3:
	(* 	Clamp State Machine 														*)
	(*		Init: TS back, collets unclamped, ejectors Retracted, Unclamped				*)
	(*		T0: Clamp Requested													*)
	(*		S1: a) Advance Tailstock to Forward Position 				 				*)
	(*			b) When collett significantly swallows part Advance Ejectors. Start Timer	*)
	(*		T1: Tailstock @ Forward Position										*)
	(*		S2: Verify  Ejectors Status of Advanced Proxes and Time Delay completed		*)
	(*		T2: Ejectors Advanced Confirmation 										*)
	(*		S3: Clamp Collet 														*)
	(*		T3: All Report Clamped PS 												*)
	(*		S4: Turn Off Postion Lag Monitoring and Set Torque Limit Value				*)
	(*		T4: Confirm Donef														*)
	(*		S5: Issue Move Velocity (in proper direction)								*)
	(*		T5: Verify Torque Value												*)
	(*		S6: REPORT CLAMPED 												*)
	IF NOT(bEnable) THEN
		bColletClamp:=FALSE;
		bColletUnclamp:=FALSE;
		bEjectorAdvance:=FALSE;
		bEjectorRetract:=FALSE;
		bTailstockAxisMove:=FALSE;
		bTailstockAxisMoveVelo:=FALSE;
		bEjectorAdvanceTON:=FALSE;
		bColletClampTON:= FALSE;
		bEjectorRetractTON:= FALSE;
		bColletUnclampTON:= FALSE;
		bTailstockAxisStop:=TRUE;
		nCurrentAction:=0;
		nClampingState:=0;
	END_IF
	IF NOT(bClampParts) THEN
		(* WE ONLY GET HERE IF THERE IS AN EXTERNAL FAULT *)
		(* Stop ALL Possible Movement *)
		bEjectorAdvance:=FALSE;
		bEjectorRetract:=FALSE;
		bColletClamp:=FALSE;
		bColletUnclamp:=FALSE;
		bEjectorAdvanceTON:=FALSE;
		bColletClampTON:= FALSE;
		bEjectorRetractTON:= FALSE;
		bColletUnclampTON:= FALSE;
		(* Stop Axis *)
		IF NOT(bTailstockAxisStop) THEN
			bTailstockAxisMove:=FALSE;
			bTailstockAxisMoveVelo:=FALSE;
			bTailstockAxisSetZero:=FALSE;
			bTailstockAxisStop:=TRUE;
		ELSIF bTailstockAxisStop AND fbTailstockAxisStop.Error THEN
			bTailstockAxisStop:=FALSE;
			(* EXIT *)
			nCurrentAction:=2;
			nClampingState:=0;
		ELSIF bTailstockAxisStop AND fbTailstockAxisStop.Done THEN
			bTailstockAxisStop:=FALSE;
			(* EXIT *)
			nCurrentAction:=2;
			nClampingState:=0;
		END_IF
	ELSE
		CASE nClampingState OF
		0:	(* Init: TS back, Parts Ready to Clamp, collets unclamped, Ejectors Retracted, Unclamped *)
			IF bClamped THEN
				nCurrentAction:=2;
			ELSIF stTailstockAxis.NcToPlc.ActPos < fTailstockBackPosition - 0.1 THEN
				nErrorID:=12;
				bError:=TRUE;
				nClampingState:=0;
				nCurrentAction:=255;
			ELSIF NOT(bColletUnclamped) THEN
				nErrorID:=13;
				bError:=TRUE;
				nClampingState:=0;
				nCurrentAction:=255;
			ELSIF NOT(stTailstockAxis.Status.Homed) THEN
				nErrorID:=1;
				bError:=TRUE;
				nClampingState:=0;
				nCurrentAction:=255;
			ELSIF NOT bTransferAtClampPosition THEN
				nErrorID:=14;
				bError:=TRUE;
				nClampingState:=0;
				nCurrentAction:=255;
			ELSIF NOT(nEjectorRetracted=7) THEN
				nErrorID:=15;
				bError:=TRUE;
				nClampingState:=0;
				nCurrentAction:=255;
			(* Begin Clamping *)
			ELSE
			(* T0: Clamp Requested *)
				(* When we are behind the transfer position we move fast to the transfer position *)
				IF (stTailstockAxis.NcToPlc.ActPos > fTailstockFrontPosition + 0.5) THEN
					nClampingState:=7;
				(* When we are at the transfer position we move at the slow speed to swallow the parts *)
				ELSE
					nClampingState:=nClampingState+1;
				END_IF
			END_IF

		1:	(* S1: a) Advance Tailstock to Forward Position
				b) When collett significantly swallows part Advance Ejectors. Start Timer *)
			IF bTailstockAxisMove AND fbTailstockAxisMoveTo.Error THEN
				bTailstockAxisMove:=FALSE;
				bTailstockAxisStop:=TRUE;
				(* Error *)
				nErrorID:=3;
				bError:=TRUE;
				nClampingState:=0;
				nCurrentAction:=255;
			(* When the Torque exceeds Max set value exit and fault *)
			ELSIF nTorqueFeedback>nClampingMaxTorqueLimit*10 THEN
				bTailstockAxisMove:=FALSE;
				bTailstockAxisStop:=TRUE;
				bError:=TRUE;
				nErrorID:=2;
				nClampingState:=0;
				nCurrentAction:=255;
			ELSIF bTailstockAxisMove AND fbTailstockAxisMoveTo.Done AND fbEjectorAdvanceTon.Q THEN
			(* T1: Tailstock @ Position *)
				bTailstockAxisMove:=FALSE;
				nClampingState:=nClampingState+1;
			ELSIF (stTailstockAxis.NcToPlc.ActPos < fTailstockFrontPosition + 8.0) THEN
			 (* S1:b) Advanced Ejectors when significantly swallowed part *)
				bEjectorAdvance:=TRUE;
			ELSE
				fTailstockAxisPosition:=fTailstockFrontPosition;
				fTailstockAxisVelocityLocal:=fTailstockAxisVelocityClamp;
				bTailstockAxisMove:=TRUE;
				(* Turn off the Retract output so the coil field can collapse before we fire other solenoid valve *)
				bEjectorRetract := FALSE;
			END_IF

		2:	(* S2: Verify  Ejectors Status of Advanced Proxes *)
			(* Fault if one of the ejectors overtraveled *)
			IF nEjectorAdvanced<7 AND nEjectorRetracted=0 AND bEjectorAdvance THEN
				(* Error *)
				nErrorID:=5;
				bError:=TRUE;
				nCurrentAction:=255;
				nClampingState:=0;
				bEjectorAdvance:=FALSE;
				bEjectorAdvanceTON:=FALSE;
			(* Basically this step gives the Ejectors a 1/2 second time delay to operate *)
			ELSIF nEjectorAdvanced=7 AND nEjectorRetracted=0 AND bEjectorAdvance  THEN
			(* T2: Ejectors Advanced *)
				nClampingState:=nClampingState+1;
			END_IF

		3:	(* S3: Clamp Collet *)
			IF bColletClamp AND fbColletClampTON.Q THEN
				(* Error *)
				nErrorID:=6;
				bError:=TRUE;
				nCurrentAction:=255;
				nClampingState:=0;
				bColletClamp:=FALSE;
				bColletClampTON:=FALSE;
			(* We look for Ejector Advanced Error in this step in case one of the Ejectors was slow *)
			ELSIF nEjectorAdvanced<7 AND nEjectorRetracted=0 AND bEjectorAdvance THEN
				(* Error *)
				nErrorID:=5;
				bError:=TRUE;
				nCurrentAction:=255;
				nClampingState:=0;
				bEjectorAdvance:=FALSE;
			ELSIF bColletClamped AND bColletClamp THEN
			(* T3: All Report Clamped *)
				bColletClampTON:=FALSE;
				nClampingState:=6;
			ELSE
				bColletUnclamp:=FALSE;
				bColletClampTON:=TRUE;
				(* Allow Solenoid to De-energize before firing Oposing Solenoid *)
				IF fbUnclampOffTON.Q THEN
					bColletClamp:=TRUE;
				END_IF
			END_IF

		(* We were unable to accomplish Torque limited move because the Ejectors overcame the Collet clamping force *)
		4:	(*S4: Turn Off Postion Lag Monitoring AND Set Torque LIMIT Value *)
			nTorqueLimit := nTorqueLimitRequest;
			IF bTogglePositionLagMonitoring AND fbTogglePositionLagMonitoring.Error THEN
				(* Error *)
				nErrorID:=20;
				bError:=TRUE;
				nCurrentAction:=255;
				nClampingState:=0;
				bTogglePositionLagMonitoring:=FALSE;
			ELSIF bTogglePositionLagMonitoring AND fbTogglePositionLagMonitoring.Done  THEN
			(* T4: Done *)
				bTogglePositionLagMonitoring:=FALSE;
				nClampingState:=nClampingState+1;
			ELSE
				bTogglePositionLagMonitoring := TRUE;
				bPositionLagMonitoiring := FALSE;
			END_IF

		5:	(* S5: Issue Move Velocity (in proper direction) *)
			IF bTailstockAxisMoveVelo AND fbTailstockAxisMoveVelo.Error
			THEN
				nVeloMoveErrorID:=fbTailstockAxisMoveVelo.ErrorID;
				bTailstockAxisMoveVelo :=FALSE;
				bTorqueLimitTimeout:=FALSE;
				bTailstockAxisStop := TRUE;
				(* Error *)
				nErrorID:=19;
				bError:=TRUE;
				nClampingState:=0;
				nCurrentAction:=255;
			ELSIF bTailstockAxisMoveVelo AND fbTorqueLimitTON.Q
			THEN
				bTailstockAxisMoveVelo :=FALSE;
				bTorqueLimitTimeout:=FALSE;
				bTailstockAxisStop := TRUE;
				(* Error *)
				nErrorID:=18;
				bError:=TRUE;
				nClampingState:=0;
				nCurrentAction:=255;
			ELSIF bTailstockAxisMoveVelo AND
				(stTailstockAxis.NcToPlc.ActPos < (fTailstockFrontPosition -0.10))
			THEN
				bTailstockAxisMoveVelo :=FALSE;
				bTorqueLimitTimeout:=FALSE;
				bTailstockAxisStop := TRUE;
				(* Error *)
				nErrorID:=17;
				bError:=TRUE;
				nClampingState:=0;
				nCurrentAction:=255;
			ELSIF bTailstockAxisMoveVelo AND (nTorqueFeedback > ( nTorqueLimitRequest - 2 )) THEN
			(* T7: In Velocity Command *)
				bTorqueLimitTimeout:=FALSE;
				bTailstockAxisMoveVelo := FALSE;
				nClampingState:=nClampingState+1;
			ELSE
				fTailstockAxisPosition:=fTailstockFrontPosition+fTailstockAxisBackOffAmount;
				fTailstockMoveVelo:=fTailstockAxisVelocity;
				bTailstockAxisMoveVelo:=TRUE;
				bTorqueLimitTimeout := TRUE;
			END_IF

		6:	(* S6: REPORT CLAMPED *)
			nClampingState:=0;
			nCurrentAction:=2;

		7:	(* Advance to Transfer position *)
			IF bTailstockAxisMove AND fbTailstockAxisMoveTo.Error THEN
				bTailstockAxisMove:=FALSE;
				bTailstockAxisStop:=TRUE;
				(* Error *)
				nErrorID:=3;
				bError:=TRUE;
				nClampingState:=0;
				nCurrentAction:=255;
			(* When the Torque exceeds Max set value exit and fault *)
			ELSIF nTorqueFeedback>nMaxFastTorqueLimit*10 THEN
				bTailstockAxisMove:=FALSE;
				bTailstockAxisStop:=TRUE;
				bError:=TRUE;
				nErrorID:=2;
				nClampingState:=0;
				nCurrentAction:=255;
			ELSIF bTailstockAxisMove AND fbTailstockAxisMoveTo.Done THEN
			(* T1: Tailstock @ Transfer Position *)
				bTailstockAxisMove:=FALSE;
				nClampingState:=1;
			ELSE
				fTailstockAxisPosition:=fTailstockBackPosition;
				fTailstockAxisVelocityLocal:=fTailstockAxisVelocity;
				bTailstockAxisMove:=TRUE;
			END_IF

		END_CASE
	END_IF

4:
	(*	Unclamp State Machine													*)
	(*		Init: All report clamped and reporting clamped								*)
	(*		T0: Unclamp Requested												*)
	(*		S1: Stop Axis															*)
	(*		T1: Done bit															*)
	(*		S2: Set Torque Back to 100%											*)
	(*		S3: Retract Tailstock Offset Amount and Retract Ejectors 						*)
	(*		T3: Tailstock @ Offset 													*)
	(*		S4: Unclamp Collets													*)
	(*		T4: Collets Unclamp PS												*)
	(*		S5: Move Tailstock to back position										*)
	(*		T5: Tailstock @ back 													*)
	(*		S6: REPORT UNCLAMPED												*)

	IF NOT(bEnable) THEN
		bColletClamp:=FALSE;
		bColletUnclamp:=FALSE;
		bEjectorAdvance:=FALSE;
		bEjectorRetract:=FALSE;
		bTailstockAxisMove:=FALSE;
		bEjectorAdvanceTON:=FALSE;
		bColletClampTON:= FALSE;
		bEjectorRetractTON:= FALSE;
		bColletUnclampTON:= FALSE;
		bTailstockAxisStop:=TRUE;
		nCurrentAction:=0;
		nUnclampingState:=0;
	END_IF
	IF NOT(bUnclampParts) THEN
		(* WE ONLY GET HERE IF THERE IS AN EXTERNAL FAULT *)
		(* Stop ALL Possible Movement *)
		bEjectorAdvance:=FALSE;
		bEjectorRetract:=FALSE;
		bColletClamp:=FALSE;
		bColletUnclamp:=FALSE;
		bEjectorAdvanceTON:=FALSE;
		bColletClampTON:= FALSE;
		bEjectorRetractTON:= FALSE;
		bColletUnclampTON:= FALSE;
		(* Stop Axis *)
		IF NOT(bTailstockAxisStop) THEN
			bTailstockAxisHome:=FALSE;
			bTailstockAxisMove:=FALSE;
			bTailstockAxisSetZero:=FALSE;
			bTailstockAxisStop:=TRUE;
		ELSIF bTailstockAxisStop AND fbTailstockAxisStop.Error THEN
			bTailstockAxisStop:=FALSE;
			(* EXIT *)
			nCurrentAction:=2;
			nUnclampingState:=0;
		ELSIF bTailstockAxisStop AND fbTailstockAxisStop.Done THEN
			bTailstockAxisStop:=FALSE;
			(* EXIT *)
			nCurrentAction:=2;
			nUnclampingState:=0;
		END_IF
	ELSE
		CASE nUnclampingState OF
		0:	(* Init: All report clamped and reporting clamped *)
			nTorqueLimit := 1000;
			IF NOT(stTailstockAxis.Status.Homed) THEN
				(* Error *)
				nErrorID:=1;
				bError:=TRUE;
				nUnclampingState:=0;
				nCurrentAction:=255;
			(* Nothing To Do Here *)
			ELSIF bUnclamped THEN
				nCurrentAction:=2;
			(* Begin Unclamping *)
			ELSE
			(* T0: Unclamp Requested *)
				nUnclampingState:=nUnclampingState+1;
			END_IF

		1: (* S1: Stop Axis *)
			IF bTailstockAxisStop AND fbTailstockAxisStop.Error THEN
				(* Error *)
				nErrorID:=7;
				bError:=TRUE;
				nUnclampingState:=0;
				nCurrentAction:=255;
				bTailstockAxisStop:=FALSE;
			ELSIF bTailstockAxisStop AND fbTailstockAxisStop.Done THEN
				bTailstockAxisStop:=FALSE;
				nUnclampingState:=nUnclampingState+1;
			ELSE
				bTailstockAxisStop:=TRUE;
			END_IF

		2: 	(* S2: Set Torque Back to 100% *)
			nTorqueLimit := 1000;
			nUnclampingState:=nUnclampingState+1;

		3:	(* S3: Retract Tailstock Offset Amount and Retract Ejectors *)
			IF bTailstockAxisMove AND fbTailstockAxisMoveTo.Error THEN
				bTailstockAxisMove:=FALSE;
				(* Error *)
				nErrorID:=9;
				bError:=TRUE;
				nUnclampingState:=0;
				nCurrentAction:=255;
			(* When the Torque exceeds Max set value exit and fault *)
			ELSIF nTorqueFeedback>nMaxFastTorqueLimit*10 THEN
				bTailstockAxisMove:=FALSE;
				bTailstockAxisStop:=TRUE;
				bError:=TRUE;
				nErrorID:=2;
				nUnclampingState:=0;
				nCurrentAction:=255;
			ELSIF bTailstockAxisMove AND fbTailstockAxisMoveTo.Done THEN
			(* T3: Tailstock Position Two *)
				bTailstockAxisMove:=FALSE;
				nUnclampingState:=nUnclampingState+1;
			ELSE
				fTailstockAxisPosition := fTailstockFrontPosition +fTailstockAxisBackOffAmount ;
				fTailstockAxisVelocityLocal:=fTailstockAxisVelocity;
				bTailstockAxisMove:=TRUE;
				bEjectorAdvance:=FALSE;
				IF fbEjectAdvOffTON.Q THEN
					bEjectorRetract:=TRUE;
				END_IF
			END_IF

		4:	(* S4: Unclamp Collets *)
			IF bColletUnclamp AND fbColletUnclampTON.Q THEN
				(* Error *)
				nErrorID:=8;
				bError:=TRUE;
				nUnclampingState:=0;
				nCurrentAction:=255;
				bColletUnclamp:=FALSE;
				bColletUnclampTON:=FALSE;
			ELSIF bColletUnclamped AND bColletUnclamp THEN
			(* T4: Collets report unclamped by PS *)
				bColletUnclampTON:=FALSE;
				nUnclampingState:=nUnclampingState+1;
			ELSE
				bColletClamp:=FALSE;
				bColletUnclampTON:=TRUE;
				IF fbClampOffTON.Q THEN
					bColletUnclamp:=TRUE;
				END_IF
			END_IF

		5: 	(* S5: Move Tailstock to back position *)
			IF bTailstockAxisMove AND fbTailstockAxisMoveTo.Error THEN
				bTailstockAxisMove:=FALSE;
				(* Error *)
				nErrorID:=9;
				bError:=TRUE;
				nUnclampingState:=0;
				nCurrentAction:=255;
			(* When the Torque exceeds Max set value exit and fault *)
			ELSIF nTorqueFeedback>nMaxFastTorqueLimit*10 THEN
				bTailstockAxisMove:=FALSE;
				bTailstockAxisStop:=TRUE;
				bError:=TRUE;
				nErrorID:=2;
				nClampingState:=0;
				nCurrentAction:=255;
			ELSIF bTailstockAxisMove AND fbTailstockAxisMoveTo.Done THEN
			(* T5: Tailstock @ Back Position *)
				bTailstockAxisMove:=FALSE;
				nUnclampingState:=0;
				nCurrentAction:=2;
		(*		nUnclampingState:=nUnclampingState+1;			*)
			ELSE
				fTailstockAxisPosition:=fTailstockBackPosition;
				fTailstockAxisVelocityLocal:=fTailstockAxisVelocity;
				bTailstockAxisMove:=TRUE;
			END_IF

		6:	(* S7: Report Unclamped *)
			nUnclampingState:=0;
			nCurrentAction:=2;

		END_CASE
	END_IF

6: (* Manual Advance Tailstock Axis *)
	IF NOT(bEnable) THEN
		bColletClamp:=FALSE;
		bColletUnclamp:=FALSE;
		bEjectorAdvance:=FALSE;
		bEjectorRetract:=FALSE;
		bTailstockAxisMove:=FALSE;
		bError:=TRUE;
		nErrorID:=0;
		nCurrentAction:=255;
	(* Transfer Axis must be home *)
	ELSIF NOT bTransferAxisHome THEN
		bError:=TRUE;
		nErrorID:=22;
		nCurrentAction:=255;
	(* Transfer Axis must be at load or unload positiion *)
	ELSIF NOT bTransferAtClampPosition THEN
		bError:=TRUE;
		nErrorID:=14;
		nCurrentAction:=255;
	(* Missing parameters for move *)
	ELSIF fTailstockBackPosition=0.0 OR fTailstockFrontPosition=0.0 THEN
		bError:=TRUE;
		nErrorID:=21;
		nCurrentAction:=255;
	(* When the Torque exceeds Max set value exit and fault *)
	(* Moving to Transfer Postion - Fast Move *)
	ELSIF ( stTailstockAxis.NcToPlc.ActPos > fTailstockBackPosition AND
		nTorqueFeedback>nMaxFastTorqueLimit*10)
	THEN
		bTailstockAxisMove:=FALSE;
		bTailstockAxisStop:=TRUE;
		bError:=TRUE;
		nErrorID:=2;
		nCurrentAction:=255;
	(* Moving to Drill Postion - Slow Move *)
	ELSIF ( stTailstockAxis.NcToPlc.ActPos > fTailstockFrontPosition) AND
	 	(stTailstockAxis.NcToPlc.ActPos < fTailstockBackPosition) AND
		(nTorqueFeedback>nClampingMaxTorqueLimit*10)
	THEN
		bTailstockAxisMove:=FALSE;
		bTailstockAxisStop:=TRUE;
		bError:=TRUE;
		nErrorID:=2;
		nCurrentAction:=255;
	(* Fault if the Cullets are not Unclamped *)
	ELSIF NOT bColletUnclamped THEN
		bError:=TRUE;
		nErrorID:=13;
		nCurrentAction:=255;
	(* We should be Good to Make the Move *)
	ELSE
		(* If we are behind the Back position we advance to the Back position *)
		IF NOT(bTailstockAxisMove) AND stTailstockAxis.NcToPlc.ActPos > fTailstockBackPosition+0.5 THEN
			bTailstockAxisMove:=TRUE;
			fTailstockAxisVelocityLocal:=fTailstockAxisVelocity;
			fTailstockAxisPosition:=fTailstockBackPosition;
		(* Else If we are behind the forward position we advance to the forward position *)
		ELSIF NOT(bTailstockAxisMove) AND stTailstockAxis.NcToPlc.ActPos > fTailstockFrontPosition+0.1 THEN
			bTailstockAxisMove:=TRUE;
			fTailstockAxisVelocityLocal:=fTailstockAxisVelocityClamp;
			fTailstockAxisPosition:=fTailstockFrontPosition;
		(* If We are already at the forward position, then Exit out of this step *)
		ELSIF stTailstockAxis.NcToPlc.ActPos <= fTailstockFrontPosition+0.1 THEN
			bTailstockAxisMove:=FALSE;
			nCurrentAction:=2;
		(* Did we have a problem? *)
		ELSIF bTailstockAxisMove AND fbTailstockAxisMoveTo.Error THEN
			bTailstockAxisMove:=FALSE;
			bError:=TRUE;
			nErrorID:=11;
			nCurrentAction:=255;
		(* Are we there yet? *)
		ELSIF bTailstockAxisMove AND fbTailstockAxisMoveTo.Done THEN
			bTailstockAxisMove:=FALSE;
			nCurrentAction:=2;
		END_IF (* Move *)
	END_IF (* Fault Checks *)

7: (* Retract Tailstock Axis *)
	IF NOT(bEnable) THEN
		bColletClamp:=FALSE;
		bColletUnclamp:=FALSE;
		bEjectorAdvance:=FALSE;
		bEjectorRetract:=FALSE;
		bTailstockAxisMove:=FALSE;
		bError:=TRUE;
		nErrorID:=0;
		nCurrentAction:=255;
	(* Transfer Axis must be home *)
	ELSIF NOT bTransferAxisHome THEN
		bError:=TRUE;
		nErrorID:=22;
		nCurrentAction:=255;
	(* Transfer Axis must be at load or unload positiion *)
	ELSIF NOT bTransferAtClampPosition THEN
		bError:=TRUE;
		nErrorID:=14;
		nCurrentAction:=255;
	(* Missing parameters for move *)
	ELSIF fTailstockBackPosition=0.0 THEN
		bError:=TRUE;
		nErrorID:=21;
		nCurrentAction:=255;
	(* When the Torque exceeds Max set value exit and fault *)
	ELSIF nTorqueFeedback>nMaxFastTorqueLimit*10 THEN
		bTailstockAxisMove:=FALSE;
		bTailstockAxisStop:=TRUE;
		bError:=TRUE;
		nErrorID:=2;
		nCurrentAction:=255;
	(* Fault if the Cullets are not Unclamped *)
	ELSIF NOT bColletUnclamped THEN
		bError:=TRUE;
		nErrorID:=13;
		nCurrentAction:=255;
	(* We should be Good to Make the Move *)
	ELSE
		(* If we are in front of  the back position we retract to the back position *)
		IF NOT(bTailstockAxisMove) AND NOT(bColletClamped)
		AND  stTailstockAxis.NcToPlc.ActPos < fTailstockBackPosition-0.1 THEN
			bTailstockAxisMove:=TRUE;
			fTailstockAxisVelocityLocal:=fTailstockAxisVelocity;
			fTailstockAxisPosition:=fTailstockBackPosition;
		(* If We are already at the back position, then Exit out of this step *)
		ELSIF stTailstockAxis.NcToPlc.ActPos >= fTailstockBackPosition-0.1 THEN
			bTailstockAxisMove:=FALSE;
			nCurrentAction:=2;
		(* Did we have a problem? *)
		ELSIF bTailstockAxisMove AND fbTailstockAxisMoveTo.Error THEN
			bTailstockAxisMove:=FALSE;
			bError:=TRUE;
			nErrorID:=11;
			nCurrentAction:=255;
		(* Can not be Clamped and Move Back *)
		ELSIF bColletClamped THEN
			bTailstockAxisMove:=FALSE;
			bError:=TRUE;
			nErrorID:=16;
			nCurrentAction:=255;
		(* Are we there yet? *)
		ELSIF bTailstockAxisMove AND fbTailstockAxisMoveTo.Done THEN
			bTailstockAxisMove:=FALSE;
			nCurrentAction:=2;
		END_IF (* Move *)
	END_IF (* Fault Checking *)

8: (* Clamp Collet *)
	bColletUnclamp:=FALSE;
	IF fbUnclampOffTON.Q THEN
		bColletClamp:=TRUE;
	END_IF
	IF NOT(bEnable) THEN
		bColletClamp:=FALSE;
		bColletUnclamp:=FALSE;
		bEjectorAdvance:=FALSE;
		bEjectorRetract:=FALSE;
		bTailstockAxisMove:=FALSE;
		bError:=TRUE;
		nErrorID:=0;
		nCurrentAction:=255;
	ELSIF bColletClamped AND NOT(bColletUnclamped) THEN
		nCurrentAction:=2;
	ELSIF fbColletClampTimeout.Q THEN
	(* TIMEOUT *)
		bError:=TRUE;
		nErrorID:=6;
		nCurrentAction:=255;
		bColletClamp:=FALSE;
	END_IF

9: (* Open Collet *)
	bColletClamp:=FALSE;
	IF fbClampOffTON.Q THEN
		bColletUnclamp:=TRUE;
	END_IF
	IF NOT(bEnable) THEN
		bColletClamp:=FALSE;
		bColletUnclamp:=FALSE;
		bEjectorAdvance:=FALSE;
		bEjectorRetract:=FALSE;
		bTailstockAxisMove:=FALSE;
		bError:=TRUE;
		nErrorID:=0;
		nCurrentAction:=255;
	ELSIF bColletUnclamped AND NOT(bColletClamped) THEN
		nCurrentAction:=2;
	ELSIF fbColletUnclampTimeout.Q THEN
	(* TIMEOUT *)
		bError:=TRUE;
		nErrorID:=8;
		nCurrentAction:=255;
		bColletUnclamp:=FALSE;
	END_IF

10: (* Advance Ejectors *)
	bEjectorRetract:=FALSE;
	IF fbEjectRetOffTON.Q THEN
		bEjectorAdvance:=TRUE;
	END_IF
	IF NOT(bEnable) THEN
		bColletClamp:=FALSE;
		bColletUnclamp:=FALSE;
		bEjectorAdvance:=FALSE;
		bEjectorRetract:=FALSE;
		bTailstockAxisMove:=FALSE;
		bError:=TRUE;
		nErrorID:=0;
		nCurrentAction:=255;
	ELSIF nEjectorRetracted=0 THEN
		nCurrentAction:=2;
	ELSIF fbEjectorAdvanceTimeout.Q THEN
	(* TIMEOUT *)
		bError:=TRUE;
		nErrorID:=4;
		nCurrentAction:=255;
		bEjectorAdvance:=FALSE;
	END_IF

11: (* Retract Ejectors *)
	bEjectorAdvance:=FALSE;
	IF fbEjectAdvOffTON.Q THEN
		bEjectorRetract:=TRUE;
	END_IF
	IF NOT(bEnable) THEN
		bColletClamp:=FALSE;
		bColletUnclamp:=FALSE;
		bEjectorAdvance:=FALSE;
		bEjectorRetract:=FALSE;
		bTailstockAxisMove:=FALSE;
		bError:=TRUE;
		nErrorID:=0;
		nCurrentAction:=255;
	ELSIF nEjectorRetracted=7 AND nEjectorAdvanced=7 THEN
		nCurrentAction:=2;
	ELSIF fbEjectorRetractTimeout.Q THEN
	(* TIMEOUT *)
		bError:=TRUE;
		nErrorID:=7;
		nCurrentAction:=255;
		bEjectorRetract:=FALSE;
	END_IF

255:	(* Faulted *)
	(* To Reset A Block Fault All Block Inputs Must Go To FALSE *)
	IF NOT(bClampParts OR bUnclampParts
		OR bManAdvanceTailstock OR bManRetractTailstock
		OR bManAdvanceCollet OR bManRetractCollet
		OR bManAdvanceEjectors OR bManRetractEjectors)
	THEN
		bError:=FALSE;
	(*	nErrorID:=0; *)
		bTailstockAxisStop:=FALSE;
		nCurrentAction:=0;
	END_IF

ELSE
	(* Unknown State Entered *)
	bError:=TRUE;
	nErrorID:=9999;
	(* GO TO FAULTED STATE *)
	nCurrentAction:=255;
END_CASE

(* What Defines Clamped *)
bClamped:= 		bColletClamp AND bEjectorAdvance AND bColletClamped AND nEjectorAdvanced=7 AND nEjectorRetracted=0
				AND (stTailstockAXIS.NcToPlc.ActPos >= fTailstockFrontPosition  - 0.1)
				AND (stTailstockAXIS.NcToPlc.ActPos <= fTailstockFrontPosition  + 0.1) ;

(* What Defines Unclamped *)
bUnclamped:=	bColletUnclamp AND bEjectorRetract AND bColletUnclamped AND nEjectorAdvanced=7
				AND (stTailstockAXIS.NcToPlc.ActPos >= fTailstockBackPosition  - 0.1)
				(* The Unclamp State Machine is expecting the Unclamp input signal to stay on for the whole cycle *)
				AND nUnclampingState=0;

(* When the Lag Monitoring is turned off and we issue a MC_Stop to the axis
	then we want to turn the Lag monitoring back on *)
IF bTogglePositionLagMonitoring AND fbTogglePositionLagMonitoring.Done AND
	NOT(nClampingState = 4)
THEN
	bTogglePositionLagMonitoring:= FALSE;
ELSIF NOT fbPositionLagMonitingStatus.Value AND bTailstockAxisStop THEN
	bTogglePositionLagMonitoring:=TRUE;
	bPositionLagMonitoiring := TRUE;
END_IF


fbTailstockAxisMoveTo(
	Execute:=bTailstockAxisMove ,
	Position:=fTailstockAxisPosition ,
	Velocity:=fTailstockAxisVelocityLocal ,
	Acceleration:=0 ,
	Deceleration:=0 ,
	Jerk:=0 ,
	BufferMode:= MC_Aborting,
	Axis:=stTailstockAxis );

fbTailstockAxisMoveVelo(
	Execute:= bTailstockAxisMoveVelo,
	Velocity:= fTailstockMoveVelo ,
	Acceleration:= 0,
	Deceleration:= 0,
	Jerk:= 0,
	Direction:= MC_Negative_Direction,
	BufferMode:= MC_Aborting,
	Options:= ,
	Axis:= stTailstockAxis,
	InVelocity=> , 
	Busy=> , 
	Active=> , 
	CommandAborted=> , 
	Error=> , 
	ErrorID=> );

fbTailstockAxisStop(
	Execute:=bTailstockAxisStop ,
	Deceleration:=0 ,
	Jerk:=0 ,
	Axis:=stTailstockAxis );

fbTogglePositionLagMonitoring(
	Execute:= bTogglePositionLagMonitoring ,
	ParameterNumber:= AxisEnPositionLagMonitoring,
	Value:= bPositionLagMonitoiring ,
	Axis:=stTailstockAxis );

fbPositionLagMonitingStatus(
	Enable:= TRUE,
	ParameterNumber:= AxisEnPositionLagMonitoring ,
	ReadMode:= READMODE_CYCLIC,
	Axis:= stTailstockAxis ,
	Valid=> ,
	Busy=> ,
	Error=> , 
	ErrorID=> , 
	Value=> );

fbColletClampTimeout(IN:=nCurrentAction=8 , PT:=t#5s);
fbColletUnclampTimeout(IN:=nCurrentAction=9 ,PT:=t#5s);
fbEjectorAdvanceTimeout(IN:=nCurrentAction=10 ,PT:=t#5s);
fbEjectorRetractTimeout(IN:=nCurrentAction=11 ,PT:=t#5s);
fbClampOffTON(IN:=NOT bColletClamp , PT:= t#100ms);
fbUnclampOffTON(IN:= NOT bColletUnclamp , PT:= t#100ms);

fbEjectorAdvanceTON(IN:=(nEjectorRetracted=0) , PT:=t#250ms);
fbEjectorRetractTON(IN:=bEjectorRetractTON, PT:=t#10s);
fbColletClampTON(IN:=bColletClampTON, PT:=t#10s);
fbColletUnclampTON(IN:=bColletUnclampTON, PT:=t#10s);
fbEjectRetOffTON(IN:=NOT bEjectorRetract, PT:=t#100ms);
fbEjectAdvOffTON(IN:=NOT bEjectorAdvance , PT:=t#100ms);

fbClampPartsRTRIG(CLK:=bClampParts);
fbUnclampPartsRTRIG(CLK:=bUnclampParts);
fbAdvanceTailstockRTRIG(CLK:=bManAdvanceTailstock);
fbRetractTailstockRTRIG(CLK:=bManRetractTailstock);
fbAdvanceColletRTRIG(CLK:=bManAdvanceCollet);
fbRetractColletRTRIG(CLK:=bManRetractCollet);
fbAdvanceEjectorsRTRIG(CLK:=bManAdvanceEjectors);
fbRetractEjectorsRTRIG(CLK:=bManRetractEjectors);
fbTorqueLimitTON(IN:= bTorqueLimitTimeout , PT:= t#30s , Q=> , ET=> );


(* ERROR CODES: *)

(* The bError bit will be on for one cycle when triggered and then will be reset the next scan in step 255 of the FB
So we want to translate into a text string from the error code *)
IF bError THEN
	CASE nErrorID OF
	01: sErrorText := '01 - Tailstock Axis lost Homed signal';
	02: sErrorText := '02 - Tailstock Thrust Exceeded Max';
	03: sErrorText := '03 - Tailstock Axis Move to Drill Failed';
	04: sErrorText := '04 - Ejector Advance Timeout';
	05: sErrorText := '05 - Missing Parts (Ejector Overtravel)';
	06: sErrorText := '06 - Collet Clamp PS Timeout';
	07: sErrorText := '07 - Ejector Retract Timeout';
	08: sErrorText := '08 - Collet Unclamp PS Timeout';
	09: sErrorText := '09 - Tailstock Axis Move Back Failed';
	10: sErrorText := '10 - Tailstock Axis Home Failed';
	11: sErrorText := '11 - Tailstock Axis Move Failed';
	12: sErrorText := '12 - Tailstock Axis not at XFR pos.';
	13: sErrorText := '13 - Unclamped P.S. is not made';
	14: sErrorText := '14 - Transfer not at Unload Position';
	15: sErrorText := '15 - Not all Ejectors report retracted';
	16: sErrorText := '16 - Must Unclamp to Retract Tailstock';
	17: sErrorText := '17 - Tailstock Axis Moved While Drilling';
	18: sErrorText := '18 - Tailstock Torque Limit Error';
	19: sErrorText := '19 - Tailstock Torque Move Error';
	20: sErrorText := '20 - Tailstock Toggle of Lag Monitoring Failed';
	21: sErrorText := '21 - Missing W Position Parameters';
	22: sErrorText := '22 - Transfer Axis Must be Homed';
	END_CASE
END_IF
END_FUNCTION_BLOCK

(* POU Function Blocks/FB_EtherCAT_Emerson, ST *)
FUNCTION_BLOCK FB_EtherCAT_Emerson
VAR_INPUT
	bRun : BOOL := FALSE;
	nRPM : UINT := 0;
	nOverride : UINT := 100;
	fRatio : LREAL := 1.0;
	bMotorDirection : BOOL := FALSE;
	bDataValid : BOOL := FALSE;
	bReset : BOOL := FALSE;
	sNetId : T_AmsNetId;
	nSlaveAddr : UINT;
END_VAR
VAR_OUTPUT
	bEnableDrive : BOOL:=FALSE;
	bUpToSpeed : BOOL := FALSE;
	bError : BOOL:=FALSE;
	nErrorID : UDINT:=0;
	stVFDInfo : Ke_VFDInfo;
END_VAR
VAR
	(*	TxPDO Variables	*)
	nMotorSpeed AT %I* : UINT := 0;
	nMotorVoltage AT %I* : UINT := 0;
	nMotorCurrent AT %I* : UDINT := 0;
	nMotorTorque AT %I* : UINT := 0;
	nMotorPower AT %I* : UINT := 0;
	nDriveStatus AT %I* : UINT := 0;
	nDCLinkVoltage AT %I* : UINT := 0;
	nOpDayCounter1 AT %I* : UINT := 0;
	nOpDayCounter2 AT %I* : UINT := 0;
	nEnergyCounter AT %I* : INT := 0;

	(*	RxPDO Variables	*)
	bRunStop	AT %Q* : BOOL := FALSE;
	bDirection AT %Q* : BOOL := FALSE;
	nSpeed AT %Q* : INT := 0;
	bDriveReset AT %Q* : BOOL := FALSE;

	(*	READ Data	*)
	arrReadData : ARRAY [0..5] OF UINT := 6(0);

	(*	Function Blocks	*)
	fbReadData0 : FB_EcCoESdoRead;
	bReadData0 : BOOL := FALSE;
	fbReadData1 : FB_EcCoESdoRead;
	bReadData1 : BOOL := FALSE;
	fbReadData2 : FB_EcCoESdoRead;
	bReadData2 : BOOL := FALSE;
	fbReadData3 : FB_EcCoESdoRead;
	bReadData3 : BOOL := FALSE;
	fbReadData4 : FB_EcCoESdoRead;
	bReadData4 : BOOL := FALSE;
	fbReadData5 : FB_EcCoESdoRead;
	bReadData5 : BOOL := FALSE;
	fbReadTimer : TON;
	bReadTimer: BOOL := FALSE;
	fbRunTrigger: R_TRIG;

	(*	Local Variables	*)
	nVFDState: Ke_VFDState := VFD_NotReady;
	nVFDRunState: Ke_VFDState := VFD_Run_Setup;
	nRPMStore: UDINT := 0;
	nNominalRPMStore: UDINT := 0;
	bDirectionStore: BOOL := FALSE;
	fRatioStore: LREAL := 1.0;
	nOverrideStore: UDINT := 100;

	fbUpToSpeedTimer: TON;
	bUpToSpeedTimer: BOOL := FALSE;
END_VAR
(*
	Read Variables Every 10 seconds when Data Valid - Bit false
	5.06, 5.07, 5.08, 5.09, 2.11, 2.21
*)
IF bDataValid THEN
	IF NOT(bReadTimer) THEN
		bReadTimer:=TRUE;
	ELSIF fbReadTimer.Q AND bReadTimer THEN
		IF
		(bReadData0 AND NOT(fbReadData0.bBusy))
		AND
		(bReadData1 AND NOT(fbReadData1.bBusy))
		AND
		(bReadData2 AND NOT(fbReadData2.bBusy))
		AND
		(bReadData3 AND NOT(fbReadData3.bBusy))
		AND
		(bReadData4 AND NOT(fbReadData4.bBusy))
		AND
		(bReadData5 AND NOT(fbReadData5.bBusy))
		THEN
			bReadData0:=FALSE;
			bReadData1:=FALSE;
			bReadData2:=FALSE;
			bReadData3:=FALSE;
			bReadData4:=FALSE;
			bReadData5:=FALSE;
			bReadTimer:=FALSE;
		ELSIF
		NOT(bReadData0 AND bReadData1 AND bReadData2 AND bReadData3 AND bReadData4 AND bReadData5)
		THEN
			bReadData0:=TRUE;
			bReadData1:=TRUE;
			bReadData2:=TRUE;
			bReadData3:=TRUE;
			bReadData4:=TRUE;
			bReadData5:=TRUE;
		END_IF
	END_IF (* Read Timer *)
END_IF (* Data Valid Check *)

(*	Convert Values	*)
IF NOT(fbReadTimer.Q) THEN
	stVFDInfo.fMotorNominalFrequency:=arrReadData[0]/10.0;
	stVFDInfo.fMotorNominalCurrent:=arrReadData[1]/100.0;
	stVFDInfo.nMotorNominalSpeed:=arrReadData[2];
	stVFDInfo.fMotorNominalVoltage:=arrReadData[3]*1.0;
	stVFDInfo.fAccelerationTime:=arrReadData[4]/10.0;
	stVFDInfo.fDecelerationTime:=arrReadData[5]/10.0;
END_IF
stVFDInfo.nMotorSpeed:=nMotorSpeed;
stVFDInfo.fMotorVoltage:=nMotorVoltage*1.0;
stVFDInfo.fMotorCurrent:=nMotorCurrent/100.0;
stVFDInfo.fMotorTorque:=nMotorTorque/10.0;
stVFDInfo.fMotorPower:=nMotorPower;
stVFDInfo.nStatusWord:=nDriveStatus;
stVFDInfo.nDCLinkVoltage:=nDCLinkVoltage;
stVFDInfo.stDayCounter.nYears:=LREAL_TO_UINT(FLOOR(nOpDayCounter1/1000.0));
stVFDInfo.stDayCounterResettable.nYears:=LREAL_TO_UINT(FLOOR(nOpDayCounter1/1000.0));
stVFDInfo.stDayCounter.nDays:=nOpDayCounter1 MOD 1000;
stVFDInfo.stDayCounterResettable.nDays:=nOpDayCounter1 MOD 1000;
stVFDInfo.stDayCounter.nHours:=LREAL_TO_UINT(FLOOR(nOpDayCounter2/100.0));
stVFDInfo.stDayCounterResettable.nHours:=LREAL_TO_UINT(FLOOR(nOpDayCounter2/100.0));
stVFDInfo.stDayCounter.nMinutes:=nOpDayCounter2 MOD 100;
stVFDInfo.stDayCounterResettable.nMinutes:=nOpDayCounter2 MOD 100;
stVFDInfo.stEnergyCounter.fEnergy:=nEnergyCounter;
stVFDInfo.stEnergyCounter.sUnits:='kWh';
stVFDInfo.stEnergyCounterResettable.fEnergy:=nEnergyCounter;
stVFDInfo.stEnergyCounterResettable.sUnits:='kWh';
stVFDInfo.bDataValid:=bDataValid;



(*	Run VFD State Machine	*)
CASE nVFDState OF
	VFD_NotReady:
		(*	We are not ready so we must have a fault *)
		IF NOT bDataValid THEN
			bError:=TRUE;
			nErrorID:=Er_DriveComm;
			bEnableDrive:=FALSE;
		ELSIF NOT(stVFDInfo.nStatusWord.0) THEN
			bError:=TRUE;
			nErrorID:=Er_DriveNotReady;
			bEnableDrive:=FALSE;
		(*	We are ready so we move on	*)
		ELSE
			bUpToSpeed:=FALSE;
			bEnableDrive:=TRUE;
			bError:=FALSE;
			nErrorID:=Er_NoError;
			nVFDState:=VFD_Ready;
		END_IF
		IF bReset AND NOT(bDriveReset) THEN
			bDriveReset:=TRUE;
		ELSIF NOT(bReset) AND bDriveReset THEN
			bDriveReset:=FALSE;
		END_IF

	VFD_Ready:
		IF bReset AND NOT(bDriveReset) THEN
			bDriveReset:=TRUE;
		ELSIF NOT(bReset) AND bDriveReset THEN
			bDriveReset:=FALSE;
		END_IF
		(*	We will go to the fault state for a Drive Fault *)
		IF NOT bDataValid  THEN
			bError:=TRUE;
			nErrorID:=Er_DriveComm;
			nVFDState:=VFD_Fault;
		ELSIF NOT(stVFDInfo.nStatusWord.0) THEN
			bError:=TRUE;
			nErrorID:=Er_DriveFaulted;
			nVFDState:=VFD_Fault;
		(*	We are ready and waiting for a run command	*)
		ELSE
			(*	Please Enable The Drive	*)
			bEnableDrive:=TRUE;
			(*	Ensure We Are Stopped	*)
			bRunStop:=FALSE;

			(*	We must first start by storing the values on the inputs. *)
			nRPMStore:=nRPM;
			nNominalRPMStore:=stVFDInfo.nMotorNominalSpeed;
			bDirectionStore:=bMotorDirection;
			fRatioStore:=fRatio;
			nOverrideStore:=nOverride;

			(*	Set Direction	*)
			bDirection:=bDirectionStore;
			(*	Set Speed	*)
			IF nNominalRPMStore>0 THEN
				nSpeed:=LREAL_TO_INT((nRPMStore*60.0*fRatioStore)/(nNominalRPMStore)*(nOverrideStore/100.0)*10);
			END_IF

			(*	We have a run request	*)
			IF fbRunTrigger.Q THEN
				bUpToSpeedTimer:=FALSE;
				nVFDRunState:=VFD_Run_AtSpeed;
				nVFDState:=VFD_Run;
			END_IF

		END_IF

	VFD_Run:
		(*	We will go to the fault state for a Drive Fault *)
		IF NOT bDataValid  THEN
			bError:=TRUE;
			nErrorID:=Er_DriveComm;
			nVFDState:=VFD_Fault;
		ELSIF NOT(stVFDInfo.nStatusWord.0) THEN
			bError:=TRUE;
			nErrorID:=Er_DriveFaulted;
			nVFDState:=VFD_Fault;
		ELSIF nRPMStore<=0 THEN
			bError:=TRUE;
			nErrorID:=Er_InvalidRPM;
			nVFDRunState:=VFD_Run_AtSpeed;
			nVFDState:=VFD_Fault;
		ELSIF fRatioStore<=0.0 THEN
			bError:=TRUE;
			nErrorID:=Er_InvalidRatio;
			nVFDRunState:=VFD_Run_AtSpeed;
			nVFDState:=VFD_Fault;
		ELSIF nOverrideStore<=0 THEN
			bError:=TRUE;
			nErrorID:=Er_InvalidOverride;
			nVFDRunState:=VFD_Run_AtSpeed;
			nVFDState:=VFD_Fault;
		ELSIF nSpeed<0 THEN
			bError:=TRUE;
			nErrorID:=Er_InvalidRPM;
			nVFDRunState:=VFD_Run_AtSpeed;
			nVFDState:=VFD_Fault;
		ELSE
			CASE nVFDRunState OF
				VFD_Run_AtSpeed:
					(*	Start the spindle	*)
					bRunStop:=TRUE;

					IF NOT(bRun) THEN
						nVFDRunState:=VFD_Run_Stop;
					ELSIF fbUpToSpeedTimer.Q AND NOT(stVFDInfo.nStatusWord.5) THEN
						bError:=TRUE;
						nErrorID:=Er_UpToSpeedTimeout;
						bUpToSpeed:=FALSE;
						nVFDState:=VFD_Fault;
					ELSIF NOT(stVFDInfo.nStatusWord.5) THEN
						bUpToSpeed:=FALSE;
					ELSIF stVFDInfo.nStatusWord.5 THEN
						(*	VFD is up to speed	*)
						bUpToSpeed:=TRUE;
						(*	Override has been requested *)
						IF NOT(nOverrideStore=nOverride)THEN
							nOverrideStore:=nOverride;
							nVFDRunState:=VFD_Run_Override;
							bUpToSpeedTimer:=FALSE;
							bUpToSpeed:=FALSE;
						END_IF
					END_IF

					(*	Monitor the up to speed signal	*)
					IF NOT(bUpToSpeedTimer) THEN
						bUpToSpeedTimer:=TRUE;
					END_IF

				VFD_Run_Override:
					nSpeed:=LREAL_TO_INT((nRPMStore*60.0*fRatioStore)/(nNominalRPMStore)*(nOverrideStore/100.0)*10);
					nVFDRunState:=VFD_Run_AtSpeed;
					bUpToSpeedTimer:=FALSE;
					bUpToSpeed:=FALSE;

				VFD_Run_Stop:
					bUpToSpeed:=FALSE;
					bUpToSpeedTimer:=FALSE;
					bRunStop:=FALSE;
					nVFDRunState:=VFD_Run_AtSpeed;
					nVFDState:=VFD_Ready;
	
			END_CASE
		END_IF

	VFD_Fault:
		bRunStop:=FALSE;
		bEnableDrive:=FALSE;
		IF bReset AND NOT(bDriveReset) THEN
			bDriveReset:=TRUE;
		ELSIF bReset AND bDriveReset THEN
			bDriveReset:=FALSE;
			bError:=FALSE;
			nErrorID:=Er_NoError;
			nVFDRunState:=VFD_Run_AtSpeed;
			nVFDState:=VFD_NotReady;
		END_IF

END_CASE




(*	5.06, 5.07, 5.08, 5.09	*)
fbReadData0(
	sNetId:=sNetId ,
	nSlaveAddr:=nSlaveAddr ,
	nSubIndex:=16#6 ,
	nIndex:=16#2005 ,
	pDstBuf:=ADR(arrReadData[0]) ,
	cbBufLen:=16#8 ,
	bExecute:=bReadData0 ,
	tTimeout:=DEFAULT_ADS_TIMEOUT ,
	bBusy=> ,
	bError=> ,
	nErrId=>
);
fbReadData1(
	sNetId:=sNetId ,
	nSlaveAddr:=nSlaveAddr ,
	nSubIndex:=16#7 ,
	nIndex:=16#2005 ,
	pDstBuf:=ADR(arrReadData[1]) ,
	cbBufLen:=16#8 ,
	bExecute:=bReadData1 ,
	tTimeout:=DEFAULT_ADS_TIMEOUT ,
	bBusy=> ,
	bError=> , 
	nErrId=>
);
fbReadData2(
	sNetId:=sNetId ,
	nSlaveAddr:=nSlaveAddr ,
	nSubIndex:=16#8 ,
	nIndex:=16#2005 ,
	pDstBuf:=ADR(arrReadData[2]) ,
	cbBufLen:=16#8 ,
	bExecute:=bReadData2 ,
	tTimeout:=DEFAULT_ADS_TIMEOUT ,
	bBusy=> ,
	bError=> , 
	nErrId=>
);
fbReadData3(
	sNetId:=sNetId ,
	nSlaveAddr:=nSlaveAddr ,
	nSubIndex:=16#9 ,
	nIndex:=16#2005 ,
	pDstBuf:=ADR(arrReadData[3]) ,
	cbBufLen:=16#8 ,
	bExecute:=bReadData3 ,
	tTimeout:=DEFAULT_ADS_TIMEOUT ,
	bBusy=> ,
	bError=> , 
	nErrId=>
);

(*	2.11	*)
fbReadData4(
	sNetId:=sNetId,
	nSlaveAddr:= nSlaveAddr ,
	nSubIndex:=16#0B ,
	nIndex:=16#2002 ,
	pDstBuf:=ADR(arrReadData[4]) ,
	cbBufLen:=16#2 ,
	bExecute:= bReadData4 ,
	tTimeout:=DEFAULT_ADS_TIMEOUT ,
	bBusy=> ,
	bError=> ,
	nErrId=>
);
(*	2.21	*)
fbReadData5(
	sNetId:=sNetId,
	nSlaveAddr:= nSlaveAddr ,
	nSubIndex:=16#15 ,
	nIndex:=16#2002 ,
	pDstBuf:=ADR(arrReadData[5]) ,
	cbBufLen:=16#2 ,
	bExecute:= bReadData5 ,
	tTimeout:=DEFAULT_ADS_TIMEOUT ,
	bBusy=> ,
	bError=> ,
	nErrId=>
);
(*	10 Second Timer	*)
fbReadTimer(
	IN:= bReadTimer ,
	PT:= t#10s ,
	Q=> ,
	ET=>
);
(*	Run Trigger	*)
fbRunTrigger(
	CLK:=bRun ,
	Q=>
);
(*	Up To Speed Timer	*)
fbUpToSpeedTimer(
	IN:=bUpToSpeedTimer ,
	PT:= LREAL_TO_TIME(stVFDInfo.fAccelerationTime*1000.0+2000.0) ,
	Q=> ,
	ET=>
);
END_FUNCTION_BLOCK

(* Visualisation MONITORING
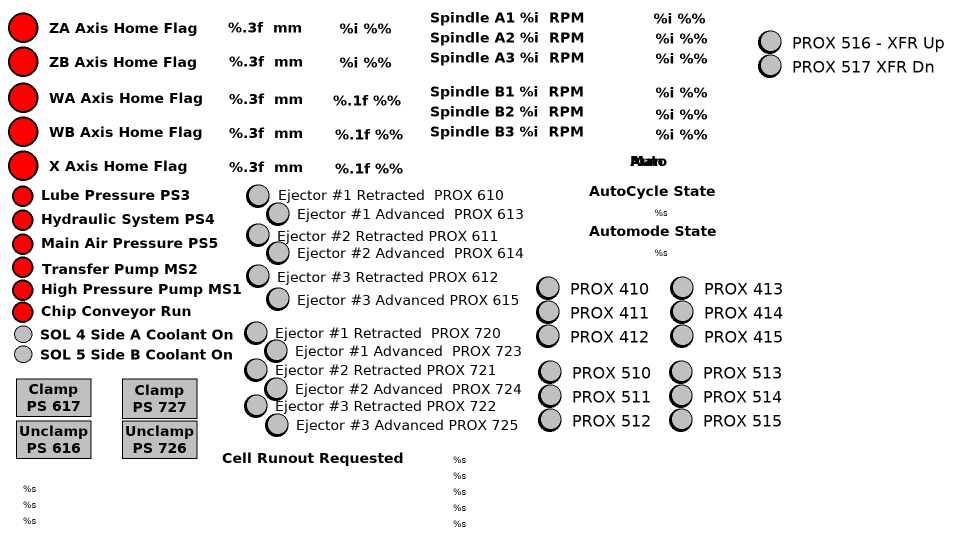
rectangle at (440,453)-(800,469): text "%s"; shows arrFaultMessage[1]; alarm colour if nFaultArrayIndex>1
rectangle at (440,469)-(800,485): text "%s"; shows arrFaultMessage[2]; alarm colour if nFaultArrayIndex>2
rectangle at (440,485)-(800,501): text "%s"; shows arrFaultMessage[3]; alarm colour if nFaultArrayIndex>3
rectangle at (10,482)-(436,498): text "%s"; shows arrFaultMessage[6]; alarm colour if nWarningArrayIndex>1
rectangle at (10,498)-(436,514): text "%s"; shows arrFaultMessage[7]; alarm colour if nWarningArrayIndex>2
rectangle at (10,514)-(436,530): text "%s"; shows arrFaultMessage[8]; alarm colour if nWarningArrayIndex>3
rectangle at (440,501)-(800,517): text "%s"; shows arrFaultMessage[4]; alarm colour if nFaultArrayIndex>4
rectangle at (440,517)-(800,533): text "%s"; shows arrFaultMessage[5]; alarm colour if nFaultArrayIndex>5
rectangle at (170,18)-(296,40): text "%.3f  mm"; shows stZAAxis.NcToPlc.ActPos
rectangle at (170,52)-(297,74): text "%.3f  mm"; shows stZBAxis.NcToPlc.ActPos
ellipse at (0,84)-(30,114): alarm colour if stWAAxis.NcToPlc.StateDWord.1
ellipse at (0,152)-(30,182): alarm colour if stUAxis.NcToPlc.StateDWord.1
rectangle at (39,87)-(199,112): text "WA Axis Home Flag"
rectangle at (39,155)-(203,180): text "X Axis Home Flag"
rectangle at (140,154)-(297,183): text "%.3f  mm"; shows stUAxis.NcToPlc.ActPos
ellipse at (0,118)-(30,148): alarm colour if stWBAxis.NcToPlc.StateDWord.1
rectangle at (39,121)-(206,146): text "WB Axis Home Flag"
rectangle at (140,120)-(297,149): text "%.3f  mm"; shows stWBAxis.NcToPlc.ActPos
rectangle at (140,86)-(297,115): text "%.3f  mm"; shows stWAAxis.NcToPlc.ActPos
ellipse at (0,14)-(30,44): alarm colour if stZAAxis.NcToPlc.StateDWord.1
rectangle at (39,17)-(199,42): text "ZA Axis Home Flag"
ellipse at (0,48)-(30,78): alarm colour if stZBAxis.NcToPlc.StateDWord.1
rectangle at (39,51)-(206,76): text "ZB Axis Home Flag"
rectangle at (420,0)-(626,38): text "Spindle A1 %i  RPM"; shows nSpindleRPM1A
rectangle at (420,20)-(626,58): text "Spindle A2 %i  RPM"; shows nSpindleRPM2A
rectangle at (420,40)-(626,78): text "Spindle A3 %i  RPM"; shows nSpindleRPM3A
rectangle at (420,74)-(626,112): text "Spindle B1 %i  RPM"; shows nSpindleRPM1B
rectangle at (420,94)-(626,132): text "Spindle B2 %i  RPM"; shows nSpindleRPM2B
rectangle at (420,114)-(626,152): text "Spindle B3 %i  RPM"; shows nSpindleRPM3B
ellipse at (4,211)-(25,232): alarm colour if bHydraulicSystemPressure
rectangle at (31,208)-(213,233): text "Hydraulic System PS4"
ellipse at (4,258)-(25,279): alarm colour if bTransferPumpMotorRunning
rectangle at (32,258)-(213,283): text "Transfer Pump MS2"
ellipse at (4,281)-(25,302): alarm colour if bHighPressureMotorRunning
rectangle at (31,278)-(232,303): text "High Pressure Pump MS1"
ellipse at (4,303)-(25,324): alarm colour if bChipConveyorMotorRunning
rectangle at (31,300)-(239,325): text "Chip Conveyor Run"
ellipse at (6,327)-(24,344): alarm colour if bACoolantSolenoid
rectangle at (30,322)-(239,350): text "SOL 4 Side A Coolant On"
ellipse at (6,347)-(24,364): alarm colour if bBCoolantSolenoid
rectangle at (30,342)-(239,370): text "SOL 5 Side B Coolant On"
ellipse at (4,235)-(25,256): alarm colour if bPneumaticSystemPressure
rectangle at (31,232)-(239,257): text "Main Air Pressure PS5"
ellipse at (4,187)-(25,208): alarm colour if bLubePressure
rectangle at (31,184)-(239,209): text "Lube Pressure PS3"
rectangle at (287,203)-(532,228): text "Ejector #1 Advanced  PROX 613"
rectangle at (287,242)-(532,267): text "Ejector #2 Advanced  PROX 614"
rectangle at (287,289)-(531,314): text "Ejector #3 Advanced PROX 615"
rectangle at (267,266)-(533,291): text "Ejector #3 Retracted PROX 612"
rectangle at (267,225)-(530,250): text "Ejector #2 Retracted PROX 611"
rectangle at (268,184)-(530,209): text "Ejector #1 Retracted  PROX 610"
ellipse at (240,186)-(261,207): alarm colour if bProx610
ellipse at (260,204)-(281,225): alarm colour if bProx613
ellipse at (240,225)-(261,246): alarm colour if bProx611
ellipse at (260,243)-(281,264): alarm colour if bProx614
ellipse at (240,266)-(261,287): alarm colour if bProx612
ellipse at (260,289)-(281,310): alarm colour if bProx615
rectangle at (264,90)-(395,114): text "%.1f %%"; shows nWAAxisThrust/10.0
rounded rectangle at (8,380)-(83,418): text "Clamp / PS 617"; alarm colour if bPS617
rounded rectangle at (8,422)-(83,460): text "Unclamp / PS 616"; alarm colour if bPS616
rectangle at (266,124)-(397,148): text "%.1f %%"; shows nWBAxisThrust/10.0
rounded rectangle at (114,380)-(189,420): text "Clamp / PS 727"; alarm colour if bPS727
rounded rectangle at (114,422)-(189,460): text "Unclamp / PS 726"; alarm colour if bPS726
rectangle at (285,340)-(530,365): text "Ejector #1 Advanced  PROX 723"
rectangle at (285,378)-(530,403): text "Ejector #2 Advanced  PROX 724"
rectangle at (286,414)-(530,439): text "Ejector #3 Advanced PROX 725"
rectangle at (265,395)-(531,420): text "Ejector #3 Retracted PROX 722"
rectangle at (265,359)-(528,384): text "Ejector #2 Retracted PROX 721"
rectangle at (265,322)-(527,347): text "Ejector #1 Retracted  PROX 720"
ellipse at (238,323)-(259,344): alarm colour if bProx720
ellipse at (258,341)-(279,362): alarm colour if bProx723
ellipse at (238,360)-(259,381): alarm colour if bProx721
ellipse at (258,379)-(279,400): alarm colour if bProx724
ellipse at (238,396)-(259,417): alarm colour if bProx722
ellipse at (259,415)-(280,436): alarm colour if bProx725
rectangle at (560,276)-(705,304): text "PROX 410"
ellipse at (530,278)-(551,299): alarm colour if bProx410
rectangle at (560,300)-(705,328): text "PROX 411"
ellipse at (530,302)-(551,323): alarm colour if bProx411
rectangle at (560,324)-(705,352): text "PROX 412"
ellipse at (530,326)-(551,347): alarm colour if bProx412
rectangle at (694,276)-(839,304): text "PROX 413"
ellipse at (664,278)-(685,299): alarm colour if bProx413
rectangle at (694,300)-(839,328): text "PROX 414"
ellipse at (664,302)-(685,323): alarm colour if bProx414
rectangle at (694,324)-(839,352): text "PROX 415"
ellipse at (664,326)-(685,347): alarm colour if bProx415
rectangle at (562,360)-(707,388): text "PROX 510"
ellipse at (532,362)-(553,383): alarm colour if bProx510
rectangle at (562,384)-(707,412): text "PROX 511"
ellipse at (532,386)-(553,407): alarm colour if bProx511
rectangle at (562,408)-(707,436): text "PROX 512"
ellipse at (532,410)-(553,431): alarm colour if bProx512
rectangle at (693,360)-(838,388): text "PROX 513"
ellipse at (663,362)-(684,383): alarm colour if bProx513
rectangle at (693,384)-(838,412): text "PROX 514"
ellipse at (663,386)-(684,407): alarm colour if bProx514
rectangle at (693,408)-(838,436): text "PROX 515"
ellipse at (663,410)-(684,431): alarm colour if bProx515
rectangle at (312,16)-(403,44): text "%i %%"; shows nServoAThrustDisplay
rectangle at (312,50)-(403,78): text "%i %%"; shows nServoBThrustDisplay
rectangle at (628,26)-(719,54): text "%i %%"; shows nSpindleLoad2ADisplay
rectangle at (628,46)-(719,74): text "%i %%"; shows nSpindleLoad3ADisplay
rectangle at (626,6)-(717,34): text "%i %%"; shows nSpindleLoad1ADisplay
rectangle at (628,102)-(719,130): text "%i %%"; shows nSpindleLoad2BDisplay
rectangle at (628,122)-(719,150): text "%i %%"; shows nSpindleLoad3BDisplay
rectangle at (628,80)-(719,108): text "%i %%"; shows nSpindleLoad1BDisplay
rectangle at (266,158)-(397,182): text "%.1f %%"; shows nUAxisThrust/10.0
rectangle at (579,180)-(739,205): text "AutoCycle State"
rectangle at (560,246)-(743,262): text "%s"; shows INT_TO_STRING(nAutoCycleStep)
rectangle at (620,150)-(680,175): text "Auto"; invisible if NOT(bMachineMode)
rectangle at (620,150)-(680,175): text "Man"; invisible if bMachineMode
rectangle at (212,447)-(427,472): text "Cell Runout Requested"; invisible if NOT(bCellRunOutRequest)
rectangle at (579,220)-(739,245): text "Automode State"
rectangle at (560,206)-(743,222): text "%s"; shows INT_TO_STRING(nAutoModeState)
rectangle at (782,30)-(971,58): text "PROX 516 - XFR Up"
ellipse at (752,32)-(773,53): alarm colour if bProx516
rectangle at (782,54)-(971,82): text "PROX 517 XFR Dn"
ellipse at (752,56)-(773,77): alarm colour if bProx517
26 more shapes without text or variables
*)
